         CASE  _response.State 
         OF
           CmdMessageState.BUFFERED : CommandBuffered := TRUE;
           CmdMessageState.DONE     : Done            := TRUE;
           CmdMessageState.ERROR    : Error           := TRUE;
         END_CASE
                
         // Done, Aborted or Error ?
         IF (_response.State >= CmdMessageState.DONE )
         THEN
           // Reset Busy flag
           Busy := FALSE;
           // Update results
           OutCmd.TargetToolNoReturn      := _response.TargetToolNoReturn;
           OutCmd.TargetFrameNoReturn     := _response.TargetFrameNoReturn;
           OutCmd.CartesianPositionReturn := _response.CartesianPositionReturn;

           // set timeout
           SetTimeout(PT := _timeoutCmd, rTimer := _timerCmd);
           // inc step counter
          _stepCmd := _stepCmd + 1; 
         END_IF
       END_IF


  02: IF ( NOT Execute)
      THEN
        Reset();
      END_IF     

ELSE
  // invalid step
  ErrorID := RobotLibraryEvents.ERR_INVALID_STEP;
END_CASE


// Reset FB
IF ( NOT Execute )
THEN
  Reset(); 
END_IF
END_METHOD

METHOD INTERNAL ParseResponsePayload : DINT
VAR_INPUT
  /// Response data
  ResponseData : RobotLibraryRecvDataFB;
  /// Timestamp
  Timestamp    : SystemTime;  
END_VAR
// Table 6-645: Received CMD payload (RC to PLC) of "CalculateCartesianPosition"
// --------------------------
// Header
// --------------------------
// Byte 00 : USINT      - ParSeq | State     
// Byte 01 : SINT       - AlarmMessageSeverity    
// Byte 02 : UINT       - AlarmMessageCode HB
// Byte 03 :            - AlarmMessageCode LB
// --------------------------
// Datablock
// --------------------------
// Byte 04 : USINT      - TargetToolNoReturn
// Byte 05 : USINT      - TargetFrameNoReturn
// Byte 06 : REAL       - Position.X  HW HB
// Byte 07 :            - Position.X  HW LB
// Byte 08 :            - Position.X  LW HB
// Byte 09 :            - Position.X  LW LB
// Byte 10 : REAL       - Position.Y  HW HB
// Byte 11 :            - Position.Y  HW LB
// Byte 12 :            - Position.Y  LW HB
// Byte 13 :            - Position.Y  LW LB
// Byte 14 : REAL       - Position.Z  HW HB
// Byte 15 :            - Position.Z  HW LB
// Byte 16 :            - Position.Z  LW HB
// Byte 17 :            - Position.Z  LW LB
// Byte 18 : REAL       - Position.Rx HW HB
// Byte 19 :            - Position.Rx HW LB
// Byte 20 :            - Position.Rx LW HB
// Byte 21 :            - Position.Rx LW LB
// Byte 22 : REAL       - Position.Ry HW HB
// Byte 23 :            - Position.Ry HW LB
// Byte 24 :            - Position.Ry LW HB
// Byte 25 :            - Position.Ry LW LB
// Byte 26 : REAL       - Position.Rz HW HB
// Byte 27 :            - Position.Rz HW LB
// Byte 28 :            - Position.Rz LW HB
// Byte 29 :            - Position.Rz LW LB
// Byte 30 : Config     - ArmConfig   LW HB
// Byte 31 :            - ArmConfig   LW LB
// Byte 32 : TurnNumber - J1 + J2     LW HB
// Byte 33 :            - J3 + J4     LW LB
// Byte 34 :            - J5 + J6     LW LB
// Byte 35 :            - E1          LW LB
// Byte 36 : REAL       - Position.E1 HW HB
// Byte 37 :            - Position.E1 HW LB
// Byte 38 :            - Position.E1 LW HB
// Byte 39 :            - Position.E1 LW LB
// Byte 40 : REAL       - Position.E2 HW HB
// Byte 41 :            - Position.E2 HW LB
// Byte 42 :            - Position.E2 LW HB
// Byte 43 :            - Position.E2 LW LB
// Byte 44 : REAL       - Position.E3 HW HB
// Byte 45 :            - Position.E3 HW LB
// Byte 46 :            - Position.E3 LW HB
// Byte 47 :            - Position.E3 LW LB
// Byte 48 : REAL       - Position.E4 HW HB
// Byte 49 :            - Position.E4 HW LB
// Byte 50 :            - Position.E4 LW HB
// Byte 51 :            - Position.E4 LW LB
// Byte 52 : REAL       - Position.E5 HW HB
// Byte 53 :            - Position.E5 HW LB
// Byte 54 :            - Position.E5 LW HB
// Byte 55 :            - Position.E5 LW LB
// Byte 56 : REAL       - Position.E6 HW HB
// Byte 57 :            - Position.E6 HW LB
// Byte 58 :            - Position.E6 LW HB
// Byte 59 :            - Position.E6 LW LB
// --------------------------
// call base implementation to parse the header from payload buffer
ResponseData.PayloadPtr := SUPER^.ParseResponsePayload(ResponseData := ResponseData, Timestamp := Timestamp);

// copy parsed header to response
_response.ParSeq               := _rspHeader.ParSeq;
_response.State                := _rspHeader.State;
_response.AlarmMessageSeverity := _rspHeader.AlarmMessageSeverity;
_response.AlarmMessageCode     := _rspHeader.AlarmMessageCode;

// Get TargetToolNoReturn
_response.TargetToolNoReturn   := ResponseData.GetUsint();
// Get TargetFrameNoReturn
_response.TargetFrameNoReturn  := ResponseData.GetUsint();
// Get CartesianPositionReturn.X
_response.CartesianPositionReturn.X := ResponseData.GetReal();
// Get CartesianPositionReturn.Y
_response.CartesianPositionReturn.Y := ResponseData.GetReal();
// Get CartesianPositionReturn.Z
_response.CartesianPositionReturn.Z := ResponseData.GetReal();
// Get CartesianPositionReturn.Rx
_response.CartesianPositionReturn.Rx := ResponseData.GetReal();
// Get CartesianPositionReturn.Ry
_response.CartesianPositionReturn.Ry := ResponseData.GetReal();
// Get CartesianPositionReturn.Rz
_response.CartesianPositionReturn.Rz := ResponseData.GetReal();
// Get CartesianPositionReturn.Config
_response.CartesianPositionReturn.Config := ResponseData.GetArmConfig();
// Get CartesianPositionReturn.TurnNumber
_response.CartesianPositionReturn.TurnNumber := ResponseData.GetTurnNumbers();
// Get CartesianPositionReturn.E1
_response.CartesianPositionReturn.E1 := ResponseData.GetReal();
// Get CartesianPositionReturn.E2
_response.CartesianPositionReturn.E2 := ResponseData.GetReal();
// Get CartesianPositionReturn.E3
_response.CartesianPositionReturn.E3 := ResponseData.GetReal();
// Get CartesianPositionReturn.E4
_response.CartesianPositionReturn.E4 := ResponseData.GetReal();
// Get CartesianPositionReturn.E5
_response.CartesianPositionReturn.E5 := ResponseData.GetReal();
// Get CartesianPositionReturn.E6
_response.CartesianPositionReturn.E6 := ResponseData.GetReal();

// Create logging
ParseResponsePayloadLog(ResponseData := ResponseData, Timestamp := Timestamp);
END_METHOD

METHOD INTERNAL ParseResponsePayloadLog
VAR_INPUT
  /// Response data
  ResponseData : RobotLibraryRecvDataFB;
  /// Timestamp
  Timestamp    : SystemTime;  
END_VAR
// Create log entry for Parameter start
CreateLogMessage      ( Timestamp   := Timestamp,
                        MessageType := MessageType.CMD,
                        Severity    := Severity.DEBUG,
                        MessageCode := 0,
                        MessageText := 'Parsed the following parameter(s) from response data:');
                        
// Create log entry for TargetToolNoReturn
CreateLogMessagePara1 ( Timestamp   := Timestamp,
                        MessageType := MessageType.CMD,
                        Severity    := Severity.DEBUG,
                        MessageCode := 0,
                        MessageText := 'Response.TargetToolNoReturn = {1}',
                        Para1       :=  USINT_TO_STRING(_response.TargetToolNoReturn));

// Create log entry for TargetFrameNoReturn
CreateLogMessagePara1 ( Timestamp   := Timestamp,
                        MessageType := MessageType.CMD,
                        Severity    := Severity.DEBUG,
                        MessageCode := 0,
                        MessageText := 'Response.TargetFrameNoReturn = {1}',
                        Para1       :=  USINT_TO_STRING(_response.TargetFrameNoReturn));

// Create log entry for CartesianPositionReturn.X
CreateLogMessagePara1 ( Timestamp   := Timestamp,
                        MessageType := MessageType.CMD,
                        Severity    := Severity.DEBUG,
                        MessageCode := 0,
                        MessageText := 'Response.CartesianPositionReturn.X = {1}',
                        Para1       :=  REAL_TO_STRING(_response.CartesianPositionReturn.X));

// Create log entry for CartesianPositionReturn.Y
CreateLogMessagePara1 ( Timestamp   := Timestamp,
                        MessageType := MessageType.CMD,
                        Severity    := Severity.DEBUG,
                        MessageCode := 0,
                        MessageText := 'Response.CartesianPositionReturn.Y = {1}',
                        Para1       :=  REAL_TO_STRING(_response.CartesianPositionReturn.Y));

// Create log entry for CartesianPositionReturn.Z
CreateLogMessagePara1 ( Timestamp   := Timestamp,
                        MessageType := MessageType.CMD,
                        Severity    := Severity.DEBUG,
                        MessageCode := 0,
                        MessageText := 'Response.CartesianPositionReturn.Z = {1}',
                        Para1       :=  REAL_TO_STRING(_response.CartesianPositionReturn.Z));

// Create log entry for CartesianPositionReturn.Rx
CreateLogMessagePara1 ( Timestamp   := Timestamp,
                        MessageType := MessageType.CMD,
                        Severity    := Severity.DEBUG,
                        MessageCode := 0,
                        MessageText := 'Response.CartesianPositionReturn.Rx = {1}',
                        Para1       :=  REAL_TO_STRING(_response.CartesianPositionReturn.Rx));

// Create log entry for CartesianPositionReturn.Ry
CreateLogMessagePara1 ( Timestamp   := Timestamp,
                        MessageType := MessageType.CMD,
                        Severity    := Severity.DEBUG,
                        MessageCode := 0,
                        MessageText := 'Response.CartesianPositionReturn.Ry = {1}',
                        Para1       :=  REAL_TO_STRING(_response.CartesianPositionReturn.Ry));

// Create log entry for CartesianPositionReturn.Rz
CreateLogMessagePara1 ( Timestamp   := Timestamp,
                        MessageType := MessageType.CMD,
                        Severity    := Severity.DEBUG,
                        MessageCode := 0,
                        MessageText := 'Response.CartesianPositionReturn.Rz = {1}',
                        Para1       :=  REAL_TO_STRING(_response.CartesianPositionReturn.Rz));

// Create log entry for CartesianPositionReturn.Config
CreateLogMessagePara1 ( Timestamp   := Timestamp,
                        MessageType := MessageType.CMD,
                        Severity    := Severity.DEBUG,
                        MessageCode := 0,
                        MessageText := 'Response.CartesianPositionReturn.Config = {1}',
                        Para1       :=  ARM_CONFIG_TO_STRING(_response.CartesianPositionReturn.Config));

// Create log entry for CartesianPositionReturn.TurnNumber.J1Turns
CreateLogMessagePara1 ( Timestamp   := Timestamp,
                        MessageType := MessageType.CMD,
                        Severity    := Severity.DEBUG,
                        MessageCode := 0,
                        MessageText := 'Response.CartesianPositionReturn.TurnNumber.J1Turns = {1}',
                        Para1       :=  SINT_TO_STRING(_response.CartesianPositionReturn.TurnNumber.J1Turns));

// Create log entry for CartesianPositionReturn.TurnNumber.J2Turns
CreateLogMessagePara1 ( Timestamp   := Timestamp,
                        MessageType := MessageType.CMD,
                        Severity    := Severity.DEBUG,
                        MessageCode := 0,
                        MessageText := 'Response.CartesianPositionReturn.TurnNumber.J2Turns = {1}',
                        Para1       :=  SINT_TO_STRING(_response.CartesianPositionReturn.TurnNumber.J2Turns));

// Create log entry for CartesianPositionReturn.TurnNumber.J3Turns
CreateLogMessagePara1 ( Timestamp   := Timestamp,
                        MessageType := MessageType.CMD,
                        Severity    := Severity.DEBUG,
                        MessageCode := 0,
                        MessageText := 'Response.CartesianPositionReturn.TurnNumber.J3Turns = {1}',
                        Para1       :=  SINT_TO_STRING(_response.CartesianPositionReturn.TurnNumber.J3Turns));

// Create log entry for CartesianPositionReturn.TurnNumber.J4Turns
CreateLogMessagePara1 ( Timestamp   := Timestamp,
                        MessageType := MessageType.CMD,
                        Severity    := Severity.DEBUG,
                        MessageCode := 0,
                        MessageText := 'Response.CartesianPositionReturn.TurnNumber.J4Turns = {1}',
                        Para1       :=  SINT_TO_STRING(_response.CartesianPositionReturn.TurnNumber.J4Turns));

// Create log entry for CartesianPositionReturn.TurnNumber.J5Turns
CreateLogMessagePara1 ( Timestamp   := Timestamp,
                        MessageType := MessageType.CMD,
                        Severity    := Severity.DEBUG,
                        MessageCode := 0,
                        MessageText := 'Response.CartesianPositionReturn.TurnNumber.J5Turns = {1}',
                        Para1       :=  SINT_TO_STRING(_response.CartesianPositionReturn.TurnNumber.J5Turns));

// Create log entry for CartesianPositionReturn.TurnNumber.J6Turns
CreateLogMessagePara1 ( Timestamp   := Timestamp,
                        MessageType := MessageType.CMD,
                        Severity    := Severity.DEBUG,
                        MessageCode := 0,
                        MessageText := 'Response.CartesianPositionReturn.TurnNumber.J6Turns = {1}',
                        Para1       :=  SINT_TO_STRING(_response.CartesianPositionReturn.TurnNumber.J6Turns));

// Create log entry for CartesianPositionReturn.TurnNumber.E1Turns
CreateLogMessagePara1 ( Timestamp   := Timestamp,
                        MessageType := MessageType.CMD,
                        Severity    := Severity.DEBUG,
                        MessageCode := 0,
                        MessageText := 'Response.CartesianPositionReturn.TurnNumber.E1Turns = {1}',
                        Para1       :=  SINT_TO_STRING(_response.CartesianPositionReturn.TurnNumber.E1Turns));

// Create log entry for CartesianPositionReturn.E1
CreateLogMessagePara1 ( Timestamp   := Timestamp,
                        MessageType := MessageType.CMD,
                        Severity    := Severity.DEBUG,
                        MessageCode := 0,
                        MessageText := 'Response.CartesianPositionReturn.E1 = {1}',
                        Para1       :=  REAL_TO_STRING(_response.CartesianPositionReturn.E1));

// Create log entry for CartesianPositionReturn.E2
CreateLogMessagePara1 ( Timestamp   := Timestamp,
                        MessageType := MessageType.CMD,
                        Severity    := Severity.DEBUG,
                        MessageCode := 0,
                        MessageText := 'Response.CartesianPositionReturn.E2 = {1}',
                        Para1       :=  REAL_TO_STRING(_response.CartesianPositionReturn.E2));

// Create log entry for CartesianPositionReturn.E3
CreateLogMessagePara1 ( Timestamp   := Timestamp,
                        MessageType := MessageType.CMD,
                        Severity    := Severity.DEBUG,
                        MessageCode := 0,
                        MessageText := 'Response.CartesianPositionReturn.E3 = {1}',
                        Para1       :=  REAL_TO_STRING(_response.CartesianPositionReturn.E3));

// Create log entry for CartesianPositionReturn.E4
CreateLogMessagePara1 ( Timestamp   := Timestamp,
                        MessageType := MessageType.CMD,
                        Severity    := Severity.DEBUG,
                        MessageCode := 0,
                        MessageText := 'Response.CartesianPositionReturn.E4 = {1}',
                        Para1       :=  REAL_TO_STRING(_response.CartesianPositionReturn.E4));

// Create log entry for CartesianPositionReturn.E5
CreateLogMessagePara1 ( Timestamp   := Timestamp,
                        MessageType := MessageType.CMD,
                        Severity    := Severity.DEBUG,
                        MessageCode := 0,
                        MessageText := 'Response.CartesianPositionReturn.E5 = {1}',
                        Para1       :=  REAL_TO_STRING(_response.CartesianPositionReturn.E5));

// Create log entry for CartesianPositionReturn.E6
CreateLogMessagePara1 ( Timestamp   := Timestamp,
                        MessageType := MessageType.CMD,
                        Severity    := Severity.DEBUG,
                        MessageCode := 0,
                        MessageText := 'Response.CartesianPositionReturn.E6 = {1}',
                        Para1       :=  REAL_TO_STRING(_response.CartesianPositionReturn.E6));
END_METHOD

METHOD PROTECTED Reset : DINT
VAR_INPUT
END_VAR
Reset := SUPER^.Reset();

Done               := FALSE;
Busy               := FALSE;
CommandBuffered    := FALSE;
END_METHOD

END_FUNCTION_BLOCK

// Library/POUs/Calculation/MC_CalculateForwardKinematic/MC_CalculateForwardKinematicFB
/// Calculate Forward Kinematic
FUNCTION_BLOCK MC_CalculateForwardKinematicFB EXTENDS RobotLibraryBaseExecuteFB
// ------------------------------------------------------------------------- 
//  SRCI Robot Library                                                
// ------------------------------------------------------------------------- 
//                                                                           
//  Object:      CalculateForwardKinematicFB                                       
//  Author:      Thorsten Brach                                                
//  Date:        2024-06-01
//
//  Description:                                              
//   
//                                                                           
//  Copyright: 
//    (C) 2024 Thorsten Brach. All rights reserved                                                                                                                                            
//             Licensed under the LGPL-3.0 license.
//                                                                           
//  Disclaimer:                                                                           
//    This project is provided without any guarantee and can be used for   
//    private and commercial purposes. Any use is at the user’s 
//    own risk and responsibility.
//
// -------------------------------------------------------------------------
VAR_INPUT
  /// Command parameter 
  ParCmd          : CalculateForwardKinematicParCmd;    
END_VAR
VAR_OUTPUT
  /// Command is transferred and confirmed by the RC
  CommandBuffered : BOOL;
  /// Command output 
  OutCmd          : CalculateForwardKinematicOutCmd;  
END_VAR

VAR
  /// internal copy of command parameter 
 _parCmd          : CalculateForwardKinematicParCmd;
  /// command data to send
 _command         : CalculateForwardKinematicSendData;
  /// response data received
 _response        : CalculateForwardKinematicRecvData;      
END_VAR

SUPER^(AxesGroup := AxesGroup);

METHOD PROTECTED CheckFunctionSupported : BOOL
VAR_IN_OUT
  /// Robot assignment of function
  AxesGroup : AxesGroup; 
END_VAR
CheckFunctionSupported := AxesGroup.InternalData.RCSupportedFunctions.CalculateForwardKinematic;

IF ( NOT CheckFunctionSupported )
THEN
  // call base implementation for set error and create log entry
  SUPER^.CheckFunctionSupported(AxesGroup := AxesGroup);
END_IF
END_METHOD

METHOD PROTECTED CheckParameterChanged : BOOL
VAR_IN_OUT
  /// Robot assignment of function
  AxesGroup    : AxesGroup; 
END_VAR
// Check ParCmd Size is > 0, because MemCmp does not work correctly with size = 0
IF (SIZEOF(ParCmd) = 0) 
THEN 
  RETURN;
END_IF

// compare memory 
_parameterChanged := ( SysDepMemCmp(pData1 := ADR(ParCmd), pData2 := ADR(_parCmd), DataLen := SIZEOF(ParCmd)) <> RobotLibraryConstants.OK );

// check parameter valid ?
_parameterValid   := CheckParameterValid( AxesGroup := AxesGroup );

IF ((  _parameterChanged        )  AND 
    (  _parameterValid          )) OR
    (  _parameterUpdateInternal )  
THEN  
  // reset internal flag for send parameter update
 _parameterUpdateInternal := FALSE;
  // update internal copy of parameters 
 _parCmd := ParCmd;
  // inc parameter sequence
 _command.ParSeq := _command.ParSeq + 1;
  // update command data  
  CommandData := CreateCommandPayload(AxesGroup := AxesGroup); // ( Access via reference to rCommandFB in ACR )
  // notify active command register 
  AxesGroup.Acyclic.ActiveCommandRegister.NotifyParameterChanged := _uniqueID;
END_IF
END_METHOD

METHOD INTERNAL CreateCommandPayload : RobotLibrarySendDataFB
VAR_IN_OUT
  /// Robot assignment of function
  AxesGroup : AxesGroup; 
END_VAR
// Table 6-632: Sent CMD payload (PLC to RC) of "CalculateForwardKinematic"
// --------------------------
// Header
// --------------------------
// Byte 00 : UINT  - Type HB     
// Byte 01 :       - Type LB    
// Byte 02 : USINT - Reserve | ExecutionMode
// Byte 03 : USINT - ParSeq  | Priority
// --------------------------
// Datablock
// --------------------------
// Byte 04 : USINT - ToolNo
// Byte 05 : USINT - FrameNo
// Byte 06 : REAL  - Position.J1  HW HB
// Byte 07 :       - Position.J1  HW LB
// Byte 08 :       - Position.J1  LW HB
// Byte 09 :       - Position.J1  LW LB
// Byte 10 : REAL  - Position.J2  HW HB
// Byte 11 :       - Position.J2  HW LB
// Byte 12 :       - Position.J2  LW HB
// Byte 13 :       - Position.J2  LW LB
// Byte 14 : REAL  - Position.J3  HW HB
// Byte 15 :       - Position.J3  HW LB
// Byte 16 :       - Position.J3  LW HB
// Byte 17 :       - Position.J3  LW LB
// Byte 18 : REAL  - Position.J4  HW HB
// Byte 19 :       - Position.J4  HW LB
// Byte 20 :       - Position.J4  LW HB
// Byte 21 :       - Position.J4  LW LB
// Byte 22 : REAL  - Position.J5  HW HB
// Byte 23 :       - Position.J5  HW LB
// Byte 24 :       - Position.J5  LW HB
// Byte 25 :       - Position.J5  LW LB
// Byte 26 : REAL  - Position.J6  HW HB
// Byte 27 :       - Position.J6  HW LB
// Byte 28 :       - Position.J6  LW HB
// Byte 29 :       - Position.J6  LW LB
// Byte 30 : REAL  - Position.E1  HW HB
// Byte 31 :       - Position.E1  HW LB
// Byte 32 :       - Position.E1  LW HB
// Byte 33 :       - Position.E1  LW LB
// Byte 34 : REAL  - Position.E2  HW HB
// Byte 35 :       - Position.E2  HW LB
// Byte 36 :       - Position.E2  LW HB
// Byte 37 :       - Position.E2  LW LB
// Byte 38 : REAL  - Position.E3  HW HB
// Byte 39 :       - Position.E3  HW LB
// Byte 40 :       - Position.E3  LW HB
// Byte 41 :       - Position.E3  LW LB
// Byte 42 : REAL  - Position.E4  HW HB
// Byte 43 :       - Position.E4  HW LB
// Byte 44 :       - Position.E4  LW HB
// Byte 45 :       - Position.E4  LW LB
// Byte 46 : REAL  - Position.E5  HW HB
// Byte 47 :       - Position.E5  HW LB
// Byte 48 :       - Position.E5  LW HB
// Byte 49 :       - Position.E5  LW LB
// Byte 50 : REAL  - Position.E6  HW HB
// Byte 51 :       - Position.E6  HW LB
// Byte 52 :       - Position.E6  LW HB
// Byte 53 :       - Position.E6  LW LB

// --------------------------
// set command parameter 
_command.CmdTyp                     :=  CmdType.CalculateForwardKinematic;
_command.ExecMode                   :=  ExecMode;
_command.ParSeq                     := _command.ParSeq;
_command.Priority                   :=  Priority;
_command.ToolNo                     := _parCmd.ToolNo;
_command.FrameNo                    := _parCmd.FrameNo;
_command.JointPosition              := _parCmd.JointPosition;

// copy command data to header
_cmdHeader := _command;
// call base implementation to copy header to payload buffer
CreateCommandPayload := SUPER^.CreateCommandPayload(AxesGroup := AxesGroup);

// add command.ToolNo
CreateCommandPayload.AddUsint(_command.ToolNo);
// add command.FrameNo
CreateCommandPayload.AddUsint(_command.FrameNo);
// add command.JointPosition.J1
CreateCommandPayload.AddReal(_command.JointPosition.J1);
// add command.JointPosition.J2
CreateCommandPayload.AddReal(_command.JointPosition.J2);
// add command.JointPosition.J3
CreateCommandPayload.AddReal(_command.JointPosition.J3);
// add command.JointPosition.J4
CreateCommandPayload.AddReal(_command.JointPosition.J4);
// add command.JointPosition.J5
CreateCommandPayload.AddReal(_command.JointPosition.J5);
// add command.JointPosition.J6
CreateCommandPayload.AddReal(_command.JointPosition.J6);
// add command.JointPosition.E1
CreateCommandPayload.AddReal(_command.JointPosition.E1);
// add command.JointPosition.E2
CreateCommandPayload.AddReal(_command.JointPosition.E2);
// add command.JointPosition.E3
CreateCommandPayload.AddReal(_command.JointPosition.E3);
// add command.JointPosition.E4
CreateCommandPayload.AddReal(_command.JointPosition.E4);
// add command.JointPosition.E5
CreateCommandPayload.AddReal(_command.JointPosition.E5);
// add command.JointPosition.E6
CreateCommandPayload.AddReal(_command.JointPosition.E6);

// Create logging
CreateCommandPayloadLog(AxesGroup := AxesGroup);
END_METHOD

METHOD INTERNAL CreateCommandPayloadLog 
VAR_IN_OUT
  /// Robot assignment of function
  AxesGroup : AxesGroup; 
END_VAR
// Create log entry for Parameter start
CreateLogMessage      ( Timestamp   := AxesGroup.InternalData.SystemTime,
                        MessageType := MessageType.CMD,
                        Severity    := Severity.DEBUG,
                        MessageCode := 0,
                        MessageText := 'Create command payload with the following parameter(s) :');

// Create log entry for ToolNo
CreateLogMessagePara1 ( Timestamp   := AxesGroup.InternalData.SystemTime,
                        MessageType := MessageType.CMD,
                        Severity    := Severity.DEBUG,
                        MessageCode := 0,
                        MessageText := 'Command.ToolNo = {1}',
                        Para1       :=  USINT_TO_STRING(_command.ToolNo));

// Create log entry for FrameNo
CreateLogMessagePara1 ( Timestamp   := AxesGroup.InternalData.SystemTime,
                        MessageType := MessageType.CMD,
                        Severity    := Severity.DEBUG,
                        MessageCode := 0,
                        MessageText := 'Command.FrameNo = {1}',
                        Para1       :=  USINT_TO_STRING(_command.FrameNo));

// Create log entry for JointPosition.J1
CreateLogMessagePara1 ( Timestamp   := AxesGroup.InternalData.SystemTime,
                        MessageType := MessageType.CMD,
                        Severity    := Severity.DEBUG,
                        MessageCode := 0,
                        MessageText := 'Command.JointPosition.J1 = {1}',
                        Para1       :=  REAL_TO_STRING(_command.JointPosition.J1));

// Create log entry for JointPosition.J2
CreateLogMessagePara1 ( Timestamp   := AxesGroup.InternalData.SystemTime,
                        MessageType := MessageType.CMD,
                        Severity    := Severity.DEBUG,
                        MessageCode := 0,
                        MessageText := 'Command.JointPosition.J2 = {1}',
                        Para1       :=  REAL_TO_STRING(_command.JointPosition.J2));

// Create log entry for JointPosition.J3
CreateLogMessagePara1 ( Timestamp   := AxesGroup.InternalData.SystemTime,
                        MessageType := MessageType.CMD,
                        Severity    := Severity.DEBUG,
                        MessageCode := 0,
                        MessageText := 'Command.JointPosition.J3 = {1}',
                        Para1       :=  REAL_TO_STRING(_command.JointPosition.J3));

// Create log entry for JointPosition.J4
CreateLogMessagePara1 ( Timestamp   := AxesGroup.InternalData.SystemTime,
                        MessageType := MessageType.CMD,
                        Severity    := Severity.DEBUG,
                        MessageCode := 0,
                        MessageText := 'Command.JointPosition.J4 = {1}',
                        Para1       :=  REAL_TO_STRING(_command.JointPosition.J4));

// Create log entry for JointPosition.J5
CreateLogMessagePara1 ( Timestamp   := AxesGroup.InternalData.SystemTime,
                        MessageType := MessageType.CMD,
                        Severity    := Severity.DEBUG,
                        MessageCode := 0,
                        MessageText := 'Command.JointPosition.J5 = {1}',
                        Para1       :=  REAL_TO_STRING(_command.JointPosition.J5));

// Create log entry for JointPosition.J6
CreateLogMessagePara1 ( Timestamp   := AxesGroup.InternalData.SystemTime,
                        MessageType := MessageType.CMD,
                        Severity    := Severity.DEBUG,
                        MessageCode := 0,
                        MessageText := 'Command.JointPosition.J6 = {1}',
                        Para1       :=  REAL_TO_STRING(_command.JointPosition.J6));

// Create log entry for JointPosition.E1
CreateLogMessagePara1 ( Timestamp   := AxesGroup.InternalData.SystemTime,
                        MessageType := MessageType.CMD,
                        Severity    := Severity.DEBUG,
                        MessageCode := 0,
                        MessageText := 'Command.JointPosition.E1 = {1}',
                        Para1       :=  REAL_TO_STRING(_command.JointPosition.E1));

// Create log entry for JointPosition.E2
CreateLogMessagePara1 ( Timestamp   := AxesGroup.InternalData.SystemTime,
                        MessageType := MessageType.CMD,
                        Severity    := Severity.DEBUG,
                        MessageCode := 0,
                        MessageText := 'Command.JointPosition.E2 = {1}',
                        Para1       :=  REAL_TO_STRING(_command.JointPosition.E2));

// Create log entry for JointPosition.E3
CreateLogMessagePara1 ( Timestamp   := AxesGroup.InternalData.SystemTime,
                        MessageType := MessageType.CMD,
                        Severity    := Severity.DEBUG,
                        MessageCode := 0,
                        MessageText := 'Command.JointPosition.E3 = {1}',
                        Para1       :=  REAL_TO_STRING(_command.JointPosition.E3));

// Create log entry for JointPosition.E4
CreateLogMessagePara1 ( Timestamp   := AxesGroup.InternalData.SystemTime,
                        MessageType := MessageType.CMD,
                        Severity    := Severity.DEBUG,
                        MessageCode := 0,
                        MessageText := 'Command.JointPosition.E4 = {1}',
                        Para1       :=  REAL_TO_STRING(_command.JointPosition.E4));

// Create log entry for JointPosition.E5
CreateLogMessagePara1 ( Timestamp   := AxesGroup.InternalData.SystemTime,
                        MessageType := MessageType.CMD,
                        Severity    := Severity.DEBUG,
                        MessageCode := 0,
                        MessageText := 'Command.JointPosition.E5 = {1}',
                        Para1       :=  REAL_TO_STRING(_command.JointPosition.E5));

// Create log entry for JointPosition.E6
CreateLogMessagePara1 ( Timestamp   := AxesGroup.InternalData.SystemTime,
                        MessageType := MessageType.CMD,
                        Severity    := Severity.DEBUG,
                        MessageCode := 0,
                        MessageText := 'Command.JointPosition.E6 = {1}',
                        Para1       :=  REAL_TO_STRING(_command.JointPosition.E6));
END_METHOD

METHOD FB_init : BOOL
VAR_INPUT
  /// if TRUE, the retain variables are initialized (warm start / cold start)
  bInitRetains : BOOL; 
  /// if TRUE, the instance afterwards gets moved into the copy code (online change)
  bInCopyCode  : BOOL;  
END_VAR
MyType := 'MC_CalculateForwardKinematicFB';

ExecMode := ExecutionMode.PARALLEL;
END_METHOD

METHOD PROTECTED OnCall
VAR_IN_OUT
  /// Robot assignment of function
  AxesGroup : AxesGroup; 
END_VAR
// call base implementation
SUPER^.OnCall(AxesGroup := AxesGroup);

CASE _stepCmd OF
  
  00:  IF ( _execute_R.Q )  
       THEN
         // Check function is supported and parameter are valid ?
         IF (( CheckFunctionSupported( AxesGroup := AxesGroup )) AND
             ( CheckParameterValid   ( AxesGroup := AxesGroup )))      
         THEN
           // set busy flag
           Busy := TRUE;
           // Reset command outputs
           SysDepMemSet(pDest := ADR(OutCmd), Value := 0, DataLen := SIZEOF(OutCmd));         
           // apply command parameter
          _parCmd := ParCmd;
           // init parameter sequence
          _command.ParSeq := 1;
           // create command data
           CommandData := CreateCommandPayload(AxesGroup := AxesGroup);
           // Add command to active command register
          _uniqueID := AxesGroup.Acyclic.ActiveCommandRegister.AddCmd( pCommandFB := ADR(THIS^ ));     
           // set timeout
           SetTimeout(PT := _timeoutCmd, rTimer := _timerCmd);
           // inc step counter
          _stepCmd := _stepCmd + 1;
         END_IF 
       END_IF
     

  01:  // Wait for responce received
       IF ( _responseReceived )
       THEN
         // reset response received flag
        _responseReceived := FALSE;

         CASE  _response.State 
         OF
           CmdMessageState.BUFFERED : CommandBuffered := TRUE;
           CmdMessageState.DONE     : Error           := TRUE;
           CmdMessageState.ERROR    : Done            := TRUE;
         END_CASE
                
         // Done, Aborted or Error ?
         IF (_response.State >= CmdMessageState.DONE )
         THEN
           // Reset Busy flag
           Busy := FALSE;
           // Update results
           OutCmd.TargetToolNoReturn      := _response.TargetToolNoReturn;
           OutCmd.TargetFrameNoReturn     := _response.TargetFrameNoReturn;
           OutCmd.CartesianPosition       := _response.CartesianPosition;

           // set timeout
           SetTimeout(PT := _timeoutCmd, rTimer := _timerCmd);
           // inc step counter
          _stepCmd := _stepCmd + 1; 
         END_IF
       END_IF


  02: IF ( NOT Execute)
      THEN
        Reset();  
      END_IF     

ELSE
  // invalid step
  ErrorID := RobotLibraryEvents.ERR_INVALID_STEP;
END_CASE


// Reset FB
IF ( NOT Execute )
THEN
  Reset();  
END_IF
END_METHOD

METHOD INTERNAL ParseResponsePayload : DINT
VAR_INPUT
  /// Response data
  ResponseData : RobotLibraryRecvDataFB;
  /// Timestamp
  Timestamp    : SystemTime;  
END_VAR
// Table 6-633: Received CMD payload (RC to PLC) of "CalculateForwardKinematic"
// --------------------------
// Header
// --------------------------
// Byte 00 : USINT      - ParSeq | State     
// Byte 01 : SINT       - AlarmMessageSeverity    
// Byte 02 : UINT       - AlarmMessageCode HB
// Byte 03 :            - AlarmMessageCode LB
// --------------------------
// Datablock
// --------------------------
// Byte 04 : USINT      - ToolNoReturn
// Byte 05 : USINT      - FrameNoReturn
// Byte 06 : REAL       - Position.X  HW HB
// Byte 07 :            - Position.X  HW LB
// Byte 08 :            - Position.X  LW HB
// Byte 09 :            - Position.X  LW LB
// Byte 10 : REAL       - Position.Y  HW HB
// Byte 11 :            - Position.Y  HW LB
// Byte 12 :            - Position.Y  LW HB
// Byte 13 :            - Position.Y  LW LB
// Byte 14 : REAL       - Position.Z  HW HB
// Byte 15 :            - Position.Z  HW LB
// Byte 16 :            - Position.Z  LW HB
// Byte 17 :            - Position.Z  LW LB
// Byte 18 : REAL       - Position.Rx HW HB
// Byte 19 :            - Position.Rx HW LB
// Byte 20 :            - Position.Rx LW HB
// Byte 21 :            - Position.Rx LW LB
// Byte 22 : REAL       - Position.Ry HW HB
// Byte 23 :            - Position.Ry HW LB
// Byte 24 :            - Position.Ry LW HB
// Byte 25 :            - Position.Ry LW LB
// Byte 26 : REAL       - Position.Rz HW HB
// Byte 27 :            - Position.Rz HW LB
// Byte 28 :            - Position.Rz LW HB
// Byte 29 :            - Position.Rz LW LB
// Byte 30 : Config     - ArmConfig   LW HB
// Byte 31 :            - ArmConfig   LW LB
// Byte 32 : TurnNumber - J1 + J2     LW HB
// Byte 33 :            - J3 + J4     LW LB
// Byte 34 :            - J5 + J6     LW LB
// Byte 35 :            - E1          LW LB
// Byte 36 : REAL       - Position.E1 HW HB
// Byte 37 :            - Position.E1 HW LB
// Byte 38 :            - Position.E1 LW HB
// Byte 39 :            - Position.E1 LW LB
// Byte 40 : REAL       - Position.E2 HW HB
// Byte 41 :            - Position.E2 HW LB
// Byte 42 :            - Position.E2 LW HB
// Byte 43 :            - Position.E2 LW LB
// Byte 44 : REAL       - Position.E3 HW HB
// Byte 45 :            - Position.E3 HW LB
// Byte 46 :            - Position.E3 LW HB
// Byte 47 :            - Position.E3 LW LB
// Byte 48 : REAL       - Position.E4 HW HB
// Byte 49 :            - Position.E4 HW LB
// Byte 50 :            - Position.E4 LW HB
// Byte 51 :            - Position.E4 LW LB
// Byte 52 : REAL       - Position.E5 HW HB
// Byte 53 :            - Position.E5 HW LB
// Byte 54 :            - Position.E5 LW HB
// Byte 55 :            - Position.E5 LW LB
// Byte 56 : REAL       - Position.E6 HW HB
// Byte 57 :            - Position.E6 HW LB
// Byte 58 :            - Position.E6 LW HB
// Byte 59 :            - Position.E6 LW LB
// --------------------------
// call base implementation to parse the header from payload buffer
ResponseData.PayloadPtr := SUPER^.ParseResponsePayload(ResponseData := ResponseData, Timestamp := Timestamp);

// copy parsed header to response
_response.ParSeq               := _rspHeader.ParSeq;
_response.State                := _rspHeader.State;
_response.AlarmMessageSeverity := _rspHeader.AlarmMessageSeverity;
_response.AlarmMessageCode     := _rspHeader.AlarmMessageCode;

// Get TargetToolNoReturn
_response.TargetToolNoReturn   := ResponseData.GetUsint();
// Get TargetFrameNoReturn
_response.TargetFrameNoReturn  := ResponseData.GetUsint();
// Get CartesianPosition.X
_response.CartesianPosition.X := ResponseData.GetReal();
// Get CartesianPosition.Y
_response.CartesianPosition.Y := ResponseData.GetReal();
// Get CartesianPosition.Z
_response.CartesianPosition.Z := ResponseData.GetReal();
// Get CartesianPosition.Rx
_response.CartesianPosition.Rx := ResponseData.GetReal();
// Get CartesianPosition.Ry
_response.CartesianPosition.Ry := ResponseData.GetReal();
// Get CartesianPosition.Rz
_response.CartesianPosition.Rz := ResponseData.GetReal();
// Get CartesianPosition.Config
_response.CartesianPosition.Config := ResponseData.GetArmConfig();
// Get CartesianPosition.TurnNumber
_response.CartesianPosition.TurnNumber := ResponseData.GetTurnNumbers();
// Get CartesianPosition.E1
_response.CartesianPosition.E1 := ResponseData.GetReal();
// Get CartesianPosition.E2
_response.CartesianPosition.E2 := ResponseData.GetReal();
// Get CartesianPosition.E3
_response.CartesianPosition.E3 := ResponseData.GetReal();
// Get CartesianPosition.E4
_response.CartesianPosition.E4 := ResponseData.GetReal();
// Get CartesianPosition.E5
_response.CartesianPosition.E5 := ResponseData.GetReal();
// Get CartesianPosition.E6
_response.CartesianPosition.E6 := ResponseData.GetReal();

// Create logging
ParseResponsePayloadLog(ResponseData := ResponseData, Timestamp := Timestamp);
END_METHOD

METHOD INTERNAL ParseResponsePayloadLog
VAR_INPUT
  /// Response data
  ResponseData : RobotLibraryRecvDataFB;
  /// Timestamp
  Timestamp    : SystemTime;  
END_VAR
// Create log entry for Parameter start
CreateLogMessage      ( Timestamp   := Timestamp,
                        MessageType := MessageType.CMD,
                        Severity    := Severity.DEBUG,
                        MessageCode := 0,
                        MessageText := 'Parsed the following parameter(s) from response data:');
                        
// Create log entry for TargetToolNoReturn
CreateLogMessagePara1 ( Timestamp   := Timestamp,
                        MessageType := MessageType.CMD,
                        Severity    := Severity.DEBUG,
                        MessageCode := 0,
                        MessageText := 'Response.TargetToolNoReturn = {1}',
                        Para1       :=  USINT_TO_STRING(_response.TargetToolNoReturn));

// Create log entry for TargetFrameNoReturn
CreateLogMessagePara1 ( Timestamp   := Timestamp,
                        MessageType := MessageType.CMD,
                        Severity    := Severity.DEBUG,
                        MessageCode := 0,
                        MessageText := 'Response.TargetFrameNoReturn = {1}',
                        Para1       :=  USINT_TO_STRING(_response.TargetFrameNoReturn));

// Create log entry for CartesianPosition.X
CreateLogMessagePara1 ( Timestamp   := Timestamp,
                        MessageType := MessageType.CMD,
                        Severity    := Severity.DEBUG,
                        MessageCode := 0,
                        MessageText := 'Response.CartesianPosition.X = {1}',
                        Para1       :=  REAL_TO_STRING(_response.CartesianPosition.X));

// Create log entry for CartesianPosition.Y
CreateLogMessagePara1 ( Timestamp   := Timestamp,
                        MessageType := MessageType.CMD,
                        Severity    := Severity.DEBUG,
                        MessageCode := 0,
                        MessageText := 'Response.CartesianPosition.Y = {1}',
                        Para1       :=  REAL_TO_STRING(_response.CartesianPosition.Y));

// Create log entry for CartesianPosition.Z
CreateLogMessagePara1 ( Timestamp   := Timestamp,
                        MessageType := MessageType.CMD,
                        Severity    := Severity.DEBUG,
                        MessageCode := 0,
                        MessageText := 'Response.CartesianPosition.Z = {1}',
                        Para1       :=  REAL_TO_STRING(_response.CartesianPosition.Z));

// Create log entry for CartesianPosition.Rx
CreateLogMessagePara1 ( Timestamp   := Timestamp,
                        MessageType := MessageType.CMD,
                        Severity    := Severity.DEBUG,
                        MessageCode := 0,
                        MessageText := 'Response.CartesianPosition.Rx = {1}',
                        Para1       :=  REAL_TO_STRING(_response.CartesianPosition.Rx));

// Create log entry for CartesianPosition.Ry
CreateLogMessagePara1 ( Timestamp   := Timestamp,
                        MessageType := MessageType.CMD,
                        Severity    := Severity.DEBUG,
                        MessageCode := 0,
                        MessageText := 'Response.CartesianPosition.Ry = {1}',
                        Para1       :=  REAL_TO_STRING(_response.CartesianPosition.Ry));

// Create log entry for CartesianPosition.Rz
CreateLogMessagePara1 ( Timestamp   := Timestamp,
                        MessageType := MessageType.CMD,
                        Severity    := Severity.DEBUG,
                        MessageCode := 0,
                        MessageText := 'Response.CartesianPosition.Rz = {1}',
                        Para1       :=  REAL_TO_STRING(_response.CartesianPosition.Rz));

// Create log entry for CartesianPosition.Config
CreateLogMessagePara1 ( Timestamp   := Timestamp,
                        MessageType := MessageType.CMD,
                        Severity    := Severity.DEBUG,
                        MessageCode := 0,
                        MessageText := 'Response.CartesianPosition.Config = {1}',
                        Para1       :=  ARM_CONFIG_TO_STRING(_response.CartesianPosition.Config));

// Create log entry for CartesianPosition.TurnNumber.J1Turns
CreateLogMessagePara1 ( Timestamp   := Timestamp,
                        MessageType := MessageType.CMD,
                        Severity    := Severity.DEBUG,
                        MessageCode := 0,
                        MessageText := 'Response.CartesianPosition.TurnNumber.J1Turns = {1}',
                        Para1       :=  SINT_TO_STRING(_response.CartesianPosition.TurnNumber.J1Turns));

// Create log entry for CartesianPosition.TurnNumber.J2Turns
CreateLogMessagePara1 ( Timestamp   := Timestamp,
                        MessageType := MessageType.CMD,
                        Severity    := Severity.DEBUG,
                        MessageCode := 0,
                        MessageText := 'Response.CartesianPosition.TurnNumber.J2Turns = {1}',
                        Para1       :=  SINT_TO_STRING(_response.CartesianPosition.TurnNumber.J2Turns));

// Create log entry for CartesianPosition.TurnNumber.J3Turns
CreateLogMessagePara1 ( Timestamp   := Timestamp,
                        MessageType := MessageType.CMD,
                        Severity    := Severity.DEBUG,
                        MessageCode := 0,
                        MessageText := 'Response.CartesianPosition.TurnNumber.J3Turns = {1}',
                        Para1       :=  SINT_TO_STRING(_response.CartesianPosition.TurnNumber.J3Turns));

// Create log entry for CartesianPosition.TurnNumber.J4Turns
CreateLogMessagePara1 ( Timestamp   := Timestamp,
                        MessageType := MessageType.CMD,
                        Severity    := Severity.DEBUG,
                        MessageCode := 0,
                        MessageText := 'Response.CartesianPosition.TurnNumber.J4Turns = {1}',
                        Para1       :=  SINT_TO_STRING(_response.CartesianPosition.TurnNumber.J4Turns));

// Create log entry for CartesianPosition.TurnNumber.J5Turns
CreateLogMessagePara1 ( Timestamp   := Timestamp,
                        MessageType := MessageType.CMD,
                        Severity    := Severity.DEBUG,
                        MessageCode := 0,
                        MessageText := 'Response.CartesianPosition.TurnNumber.J5Turns = {1}',
                        Para1       :=  SINT_TO_STRING(_response.CartesianPosition.TurnNumber.J5Turns));

// Create log entry for CartesianPosition.TurnNumber.J6Turns
CreateLogMessagePara1 ( Timestamp   := Timestamp,
                        MessageType := MessageType.CMD,
                        Severity    := Severity.DEBUG,
                        MessageCode := 0,
                        MessageText := 'Response.CartesianPosition.TurnNumber.J6Turns = {1}',
                        Para1       :=  SINT_TO_STRING(_response.CartesianPosition.TurnNumber.J6Turns));

// Create log entry for CartesianPosition.TurnNumber.E1Turns
CreateLogMessagePara1 ( Timestamp   := Timestamp,
                        MessageType := MessageType.CMD,
                        Severity    := Severity.DEBUG,
                        MessageCode := 0,
                        MessageText := 'Response.CartesianPosition.TurnNumber.E1Turns = {1}',
                        Para1       :=  SINT_TO_STRING(_response.CartesianPosition.TurnNumber.E1Turns));

// Create log entry for CartesianPosition.E1
CreateLogMessagePara1 ( Timestamp   := Timestamp,
                        MessageType := MessageType.CMD,
                        Severity    := Severity.DEBUG,
                        MessageCode := 0,
                        MessageText := 'Response.CartesianPosition.E1 = {1}',
                        Para1       :=  REAL_TO_STRING(_response.CartesianPosition.E1));

// Create log entry for CartesianPosition.E2
CreateLogMessagePara1 ( Timestamp   := Timestamp,
                        MessageType := MessageType.CMD,
                        Severity    := Severity.DEBUG,
                        MessageCode := 0,
                        MessageText := 'Response.CartesianPosition.E2 = {1}',
                        Para1       :=  REAL_TO_STRING(_response.CartesianPosition.E2));

// Create log entry for CartesianPosition.E3
CreateLogMessagePara1 ( Timestamp   := Timestamp,
                        MessageType := MessageType.CMD,
                        Severity    := Severity.DEBUG,
                        MessageCode := 0,
                        MessageText := 'Response.CartesianPosition.E3 = {1}',
                        Para1       :=  REAL_TO_STRING(_response.CartesianPosition.E3));

// Create log entry for CartesianPosition.E4
CreateLogMessagePara1 ( Timestamp   := Timestamp,
                        MessageType := MessageType.CMD,
                        Severity    := Severity.DEBUG,
                        MessageCode := 0,
                        MessageText := 'Response.CartesianPosition.E4 = {1}',
                        Para1       :=  REAL_TO_STRING(_response.CartesianPosition.E4));

// Create log entry for CartesianPosition.E5
CreateLogMessagePara1 ( Timestamp   := Timestamp,
                        MessageType := MessageType.CMD,
                        Severity    := Severity.DEBUG,
                        MessageCode := 0,
                        MessageText := 'Response.CartesianPosition.E5 = {1}',
                        Para1       :=  REAL_TO_STRING(_response.CartesianPosition.E5));

// Create log entry for CartesianPosition.E6
CreateLogMessagePara1 ( Timestamp   := Timestamp,
                        MessageType := MessageType.CMD,
                        Severity    := Severity.DEBUG,
                        MessageCode := 0,
                        MessageText := 'Response.CartesianPosition.E6 = {1}',
                        Para1       :=  REAL_TO_STRING(_response.CartesianPosition.E6));
END_METHOD

METHOD PROTECTED Reset : DINT
VAR_INPUT
END_VAR
Reset := SUPER^.Reset();

Done               := FALSE;
Busy               := FALSE;
CommandBuffered    := FALSE;
END_METHOD

END_FUNCTION_BLOCK

// Library/POUs/Calculation/MC_CalculateFrame/MC_CalculateFrameFB
/// Calculate frame with three-point method
FUNCTION_BLOCK MC_CalculateFrameFB EXTENDS RobotLibraryBaseExecuteFB
// ------------------------------------------------------------------------- 
//  SRCI Robot Library                                                
// ------------------------------------------------------------------------- 
//                                                                           
//  Object:      CalculateFrameFB                                       
//  Author:      Thorsten Brach                                                
//  Date:        2024-06-09
//
//  Description:                                              
//   
//                                                                           
//  Copyright: 
//    (C) 2024 Thorsten Brach. All rights reserved                                                                                                                                            
//             Licensed under the LGPL-3.0 license.
//                                                                           
//  Disclaimer:                                                                           
//    This project is provided without any guarantee and can be used for   
//    private and commercial purposes. Any use is at the user’s 
//    own risk and responsibility.
//
// -------------------------------------------------------------------------
VAR_INPUT
  /// command parameter 
  ParCmd          : CalculateFrameParCmd;
END_VAR
VAR_OUTPUT
  /// Command is transferred and confirmed by the RC
  CommandBuffered : BOOL;
  /// Command output 
  OutCmd          : CalculateFrameOutCmd;    
END_VAR

VAR
  /// internal copy of command parameter 
 _parCmd          : CalculateFrameParCmd;
  /// command data to send
 _command         : CalculateFrameSendData;
  /// response data received
 _response        : CalculateFrameRecvData;      
  /// Incremented with each position of the input parameter "PositionsArray" sent from the PLC to the RC.
  /// Default: 0
 _dataIndex       : USINT;
  /// Set TRUE by the client, when according to the user selected "Mode" the final position of the input parameter "PositionsArray" is sent to the RC.
  /// Default: FALSE
 _dataComplete    : BOOL;
END_VAR

SUPER^(AxesGroup := AxesGroup);

METHOD PROTECTED CheckFunctionSupported : BOOL
VAR_IN_OUT
  /// Robot assignment of function
  AxesGroup : AxesGroup; 
END_VAR
CheckFunctionSupported := AxesGroup.InternalData.RCSupportedFunctions.CalculateFrame;

IF ( NOT CheckFunctionSupported )
THEN
  // call base implementation for set error and create log entry
  SUPER^.CheckFunctionSupported(AxesGroup := AxesGroup);
END_IF
END_METHOD

METHOD PROTECTED CheckParameterChanged : BOOL
VAR_IN_OUT
  /// Robot assignment of function
  AxesGroup    : AxesGroup; 
END_VAR
// Check ParCmd Size is > 0, because MemCmp does not work correctly with size = 0
IF (SIZEOF(ParCmd) = 0) 
THEN 
  RETURN;
END_IF

// compare memory 
_parameterChanged := ( SysDepMemCmp(pData1 := ADR(ParCmd), pData2 := ADR(_parCmd), DataLen := SIZEOF(ParCmd)) <> RobotLibraryConstants.OK );

// check parameter valid ?
_parameterValid   := CheckParameterValid( AxesGroup := AxesGroup );

IF ((  _parameterChanged        )  AND 
    (  _parameterValid          )) OR
    (  _parameterUpdateInternal )  
THEN  
  // reset internal flag for send parameter update
 _parameterUpdateInternal := FALSE;
  // update internal copy of parameters 
 _parCmd := ParCmd;
  // inc parameter sequence
 _command.ParSeq := _command.ParSeq + 1;
  // update command data  
  CommandData := CreateCommandPayload(AxesGroup := AxesGroup); // ( Access via reference to rCommandFB in ACR )
  // notify active command register 
  AxesGroup.Acyclic.ActiveCommandRegister.NotifyParameterChanged := _uniqueID;
END_IF
END_METHOD

METHOD INTERNAL CreateCommandPayload : RobotLibrarySendDataFB
VAR_IN_OUT
  /// Robot assignment of function
  AxesGroup : AxesGroup; 
END_VAR
// Table 6-656: Sent CMD payload (PLC to RC) of "CalculateFrame"
// --------------------------
// Header
// --------------------------
// Byte 00 : UINT       - Type HB     
// Byte 01 :            - Type LB    
// Byte 02 : USINT      - Reserve | ExecutionMode
// Byte 03 : USINT      - ParSeq  | Priority
// --------------------------
// Datablock
// --------------------------
// Byte 04 : USIN       - DataIndex
// Byte 05 : BOOL       - DataComplete
// Byte 06 : BYTE       - Reserve
// Byte 07 : USINT      - FrameNo
// Byte 08 : USINT      - ReferenceFrame
// Byte 09 : SINT       - Mode
// Byte 10 : REAL       - Position X  HW HB
// Byte 11 :            - Position X  HW LB
// Byte 12 :            - Position X  LW HB
// Byte 13 :            - Position X  LW LB
// Byte 14 : REAL       - Position Y  HW HB
// Byte 15 :            - Position Y  HW LB
// Byte 16 :            - Position Y  LW HB
// Byte 17 :            - Position Y  LW LB
// Byte 18 : REAL       - Position Z  HW HB
// Byte 19 :            - Position Z  HW LB
// Byte 20 :            - Position Z  LW HB
// Byte 21 :            - Position Z  LW LB
// Byte 22 : REAL       - Position Rx HW HB
// Byte 23 :            - Position Rx HW LB
// Byte 24 :            - Position Rx LW HB
// Byte 25 :            - Position Rx LW LB
// Byte 26 : REAL       - Position Ry HW HB
// Byte 27 :            - Position Ry HW LB
// Byte 28 :            - Position Ry LW HB
// Byte 29 :            - Position Ry LW LB
// Byte 30 : REAL       - Position Rz HW HB
// Byte 31 :            - Position Rz HW LB
// Byte 32 :            - Position Rz LW HB
// Byte 33 :            - Position Rz LW LB
// Byte 34 : Config     - ArmConfig   LW HB
// Byte 35 :            - ArmConfig   LW LB
// Byte 36 : TurnNumber - J1 + J2     LW HB
// Byte 37 :            - J3 + J4     LW LB
// Byte 38 :            - J5 + J6     LW LB
// Byte 39 :            - E1          LW LB
// Byte 40 : REAL       - Position E1 HW HB
// Byte 41 :            - Position E1 HW LB
// Byte 42 :            - Position E1 LW HB
// Byte 43 :            - Position E1 LW LB
// Byte 44 : REAL       - Position E2 HW HB
// Byte 45 :            - Position E2 HW LB
// Byte 46 :            - Position E2 LW HB
// Byte 47 :            - Position E2 LW LB
// Byte 48 : REAL       - Position E3 HW HB
// Byte 49 :            - Position E3 HW LB
// Byte 50 :            - Position E3 LW HB
// Byte 51 :            - Position E3 LW LB
// Byte 52 : REAL       - Position E4 HW HB
// Byte 53 :            - Position E4 HW LB
// Byte 54 :            - Position E4 LW HB
// Byte 55 :            - Position E4 LW LB
// Byte 56 : REAL       - Position E5 HW HB
// Byte 57 :            - Position E5 HW LB
// Byte 58 :            - Position E5 LW HB
// Byte 59 :            - Position E5 LW LB
// Byte 60 : REAL       - Position E6 HW HB
// Byte 61 :            - Position E6 HW LB
// Byte 62 :            - Position E6 LW HB
// Byte 63 :            - Position E6 LW LB
// --------------------------
// set command parameter 
_command.CmdTyp         :=  CmdType.CalculateFrame;
_command.ExecMode       :=  ExecMode;
_command.ParSeq         := _command.ParSeq;
_command.Priority       :=  Priority;
_command.FrameNo        := _parCmd.FrameNo;
_command.DataIndex      := _dataIndex;
_command.DataComplete.0 := _dataComplete;
_command.Reserve        := 0;
_command.FrameNo        := _parCmd.FrameNo;                 
_command.ReferenceFrame := _parCmd.ReferenceFrame;
_command.Mode           := _parCmd.Mode;

CASE _parCmd.Mode OF
  
  FrameCalculationMode.THREE_POINT_METHOD :

    CASE _dataIndex OF
      
      1: _command.Position := _parCmd.Origin;
      2: _command.Position := _parCmd.Position_X;
      3: _command.Position := _parCmd.Position_XY;
      
    END_CASE
  
  FrameCalculationMode.FOUR_POINT_METHOD  :

    CASE _dataIndex OF
      
      1: _command.Position := _parCmd.Origin;
      2: _command.Position := _parCmd.Position_X;
      3: _command.Position := _parCmd.Position_XY;
      4: _command.Position := _parCmd.OriginShift;      

    END_CASE
  
  FrameCalculationMode.ONE_POINT_METHOD   :
  
   _command.Position := _parCmd.Origin;

END_CASE

// copy command data to header
_cmdHeader := _command;
// call base implementation to copy header to payload buffer
CreateCommandPayload := SUPER^.CreateCommandPayload(AxesGroup := AxesGroup);

// add command.DataIndex
CreateCommandPayload.AddUsint(_command.DataIndex);
// add command.DataComplete
CreateCommandPayload.AddByte(_command.DataComplete);
// add command.Reserve
CreateCommandPayload.AddByte(_command.Reserve);
// add command.FrameNo
CreateCommandPayload.AddUsint(_command.FrameNo);
// add command.ReferenceFrame
CreateCommandPayload.AddUsint(_command.ReferenceFrame);
// add command.Mode
CreateCommandPayload.AddSint(_command.Mode);
// add command.Position.X
CreateCommandPayload.AddReal(_command.Position.X);
// add command.Position.Y
CreateCommandPayload.AddReal(_command.Position.Y);
// add command.Position.Z
CreateCommandPayload.AddReal(_command.Position.Z);
// add command.Position.Rx
CreateCommandPayload.AddReal(_command.Position.Rx);
// add command.Position.Ry
CreateCommandPayload.AddReal(_command.Position.Ry);
// add command.Position.Rz
CreateCommandPayload.AddReal(_command.Position.Rz);
// add command.Position.Config
CreateCommandPayload.AddArmConfig(_command.Position.Config);
// add command.Position.TurnNumber
CreateCommandPayload.AddTurnNumber(_command.Position.TurnNumber);
// add command.Position.E1
CreateCommandPayload.AddReal(_command.Position.E1);
// add command.Position.E2
CreateCommandPayload.AddReal(_command.Position.E2);
// add command.Position.E3
CreateCommandPayload.AddReal(_command.Position.E3);
// add command.Position.E4
CreateCommandPayload.AddReal(_command.Position.E4);
// add command.Position.E5
CreateCommandPayload.AddReal(_command.Position.E5);
// add command.Position.E6
CreateCommandPayload.AddReal(_command.Position.E6);

// Create logging
CreateCommandPayloadLog(AxesGroup := AxesGroup);
END_METHOD

METHOD INTERNAL CreateCommandPayloadLog 
VAR_IN_OUT
  /// Robot assignment of function
  AxesGroup : AxesGroup; 
END_VAR
// Create log entry for Parameter start
CreateLogMessage      ( Timestamp   := AxesGroup.InternalData.SystemTime,
                        MessageType := MessageType.CMD,
                        Severity    := Severity.DEBUG,
                        MessageCode := 0,
                        MessageText := 'Create command payload with the following parameter(s) :');

// Create log entry for DataIndex
CreateLogMessagePara1 ( Timestamp   := AxesGroup.InternalData.SystemTime,
                        MessageType := MessageType.CMD,
                        Severity    := Severity.DEBUG,
                        MessageCode := 0,
                        MessageText := 'Command.DataIndex = {1}',
                        Para1       :=  USINT_TO_STRING(_command.DataIndex));

// Create log entry for DataComplete
CreateLogMessagePara1 ( Timestamp   := AxesGroup.InternalData.SystemTime,
                        MessageType := MessageType.CMD,
                        Severity    := Severity.DEBUG,
                        MessageCode := 0,
                        MessageText := 'Command.DataComplete = {1}',
                        Para1       :=  BYTE_TO_STRING(_command.DataComplete));

// Create log entry for Reserve
CreateLogMessagePara1 ( Timestamp   := AxesGroup.InternalData.SystemTime,
                        MessageType := MessageType.CMD,
                        Severity    := Severity.DEBUG,
                        MessageCode := 0,
                        MessageText := 'Command.Reserve = {1}',
                        Para1       :=  BYTE_TO_STRING(_command.Reserve));

// Create log entry for FrameNo
CreateLogMessagePara1 ( Timestamp   := AxesGroup.InternalData.SystemTime,
                        MessageType := MessageType.CMD,
                        Severity    := Severity.DEBUG,
                        MessageCode := 0,
                        MessageText := 'Command.FrameNo = {1}',
                        Para1       :=  USINT_TO_STRING(_command.FrameNo));

// Create log entry for ReferenceFrame
CreateLogMessagePara1 ( Timestamp   := AxesGroup.InternalData.SystemTime,
                        MessageType := MessageType.CMD,
                        Severity    := Severity.DEBUG,
                        MessageCode := 0,
                        MessageText := 'Command.ReferenceFrame = {1}',
                        Para1       :=  USINT_TO_STRING(_command.ReferenceFrame));

// Create log entry for Mode
CreateLogMessagePara1 ( Timestamp   := AxesGroup.InternalData.SystemTime,
                        MessageType := MessageType.CMD,
                        Severity    := Severity.DEBUG,
                        MessageCode := 0,
                        MessageText := 'Command.Mode = {1}',
                        Para1       :=  FRAME_CALCULATION_MODE_TO_STRING(_command.Mode));


// Create log entry for Position.X
CreateLogMessagePara1 ( Timestamp   := AxesGroup.InternalData.SystemTime,
                        MessageType := MessageType.CMD,
                        Severity    := Severity.DEBUG,
                        MessageCode := 0,
                        MessageText := 'Command.Position.X = {1}',
                        Para1       :=  REAL_TO_STRING(_command.Position.X));

// Create log entry for Position.Y
CreateLogMessagePara1 ( Timestamp   := AxesGroup.InternalData.SystemTime,
                        MessageType := MessageType.CMD,
                        Severity    := Severity.DEBUG,
                        MessageCode := 0,
                        MessageText := 'Command.Position.Y = {1}',
                        Para1       :=  REAL_TO_STRING(_command.Position.Y));

// Create log entry for Position.Z
CreateLogMessagePara1 ( Timestamp   := AxesGroup.InternalData.SystemTime,
                        MessageType := MessageType.CMD,
                        Severity    := Severity.DEBUG,
                        MessageCode := 0,
                        MessageText := 'Command.Position.Z = {1}',
                        Para1       :=  REAL_TO_STRING(_command.Position.Z));

// Create log entry for Position.Rx
CreateLogMessagePara1 ( Timestamp   := AxesGroup.InternalData.SystemTime,
                        MessageType := MessageType.CMD,
                        Severity    := Severity.DEBUG,
                        MessageCode := 0,
                        MessageText := 'Command.Position.Rx = {1}',
                        Para1       :=  REAL_TO_STRING(_command.Position.Rx));

// Create log entry for Position.Ry
CreateLogMessagePara1 ( Timestamp   := AxesGroup.InternalData.SystemTime,
                        MessageType := MessageType.CMD,
                        Severity    := Severity.DEBUG,
                        MessageCode := 0,
                        MessageText := 'Command.Position.Ry = {1}',
                        Para1       :=  REAL_TO_STRING(_command.Position.Ry));

// Create log entry for Position.Rz
CreateLogMessagePara1 ( Timestamp   := AxesGroup.InternalData.SystemTime,
                        MessageType := MessageType.CMD,
                        Severity    := Severity.DEBUG,
                        MessageCode := 0,
                        MessageText := 'Command.Position.Rz = {1}',
                        Para1       :=  REAL_TO_STRING(_command.Position.Rz));

// Create log entry for Position.Config
CreateLogMessagePara1 ( Timestamp   := AxesGroup.InternalData.SystemTime,
                        MessageType := MessageType.CMD,
                        Severity    := Severity.DEBUG,
                        MessageCode := 0,
                        MessageText := 'Command.Position.Config = {1}',
                        Para1       :=  ARM_CONFIG_TO_STRING(_command.Position.Config));

// Create log entry for Position.TurnNumber[0]
CreateLogMessagePara1 ( Timestamp   := AxesGroup.InternalData.SystemTime,
                        MessageType := MessageType.CMD,
                        Severity    := Severity.DEBUG,
                        MessageCode := 0,
                        MessageText := 'Command.Position.TurnNumber[0] = {1}',
                        Para1       :=  BYTE_TO_STRING(CombineHalfSints(HalfSintHi := _command.Position.TurnNumber.J2Turns, 
                                                                        HalfSintLo := _command.Position.TurnNumber.J1Turns)));

// Create log entry for Position.TurnNumber[1]
CreateLogMessagePara1 ( Timestamp   := AxesGroup.InternalData.SystemTime,
                        MessageType := MessageType.CMD,
                        Severity    := Severity.DEBUG,
                        MessageCode := 0,
                        MessageText := 'Command.Position.TurnNumber[1] = {1}',
                        Para1       :=  BYTE_TO_STRING(CombineHalfSints(HalfSintHi := _command.Position.TurnNumber.J4Turns, 
                                                                        HalfSintLo := _command.Position.TurnNumber.J3Turns)));

// Create log entry for Position.TurnNumber[2]
CreateLogMessagePara1 ( Timestamp   := AxesGroup.InternalData.SystemTime,
                        MessageType := MessageType.CMD,
                        Severity    := Severity.DEBUG,
                        MessageCode := 0,
                        MessageText := 'Command.Position.TurnNumber[2] = {1}',
                        Para1       :=  BYTE_TO_STRING(CombineHalfSints(HalfSintHi := _command.Position.TurnNumber.J6Turns, 
                                                                        HalfSintLo := _command.Position.TurnNumber.J5Turns)));

// Create log entry for Position.TurnNumber[3]
CreateLogMessagePara1 ( Timestamp   := AxesGroup.InternalData.SystemTime,
                        MessageType := MessageType.CMD,
                        Severity    := Severity.DEBUG,
                        MessageCode := 0,
                        MessageText := 'Command.Position.TurnNumber[3] = {1}',
                        Para1       :=  SINT_TO_STRING(_command.Position.TurnNumber.E1Turns));

// Create log entry for Position.E1
CreateLogMessagePara1 ( Timestamp   := AxesGroup.InternalData.SystemTime,
                        MessageType := MessageType.CMD,
                        Severity    := Severity.DEBUG,
                        MessageCode := 0,
                        MessageText := 'Command.Position.E1 = {1}',
                        Para1       :=  REAL_TO_STRING(_command.Position.E1));

// Create log entry for Position.E2
CreateLogMessagePara1 ( Timestamp   := AxesGroup.InternalData.SystemTime,
                        MessageType := MessageType.CMD,
                        Severity    := Severity.DEBUG,
                        MessageCode := 0,
                        MessageText := 'Command.Position.E2 = {1}',
                        Para1       :=  REAL_TO_STRING(_command.Position.E2));

// Create log entry for Position.E3
CreateLogMessagePara1 ( Timestamp   := AxesGroup.InternalData.SystemTime,
                        MessageType := MessageType.CMD,
                        Severity    := Severity.DEBUG,
                        MessageCode := 0,
                        MessageText := 'Command.Position.E3 = {1}',
                        Para1       :=  REAL_TO_STRING(_command.Position.E3));

// Create log entry for Position.E4
CreateLogMessagePara1 ( Timestamp   := AxesGroup.InternalData.SystemTime,
                        MessageType := MessageType.CMD,
                        Severity    := Severity.DEBUG,
                        MessageCode := 0,
                        MessageText := 'Command.Position.E4 = {1}',
                        Para1       :=  REAL_TO_STRING(_command.Position.E4));

// Create log entry for Position.E5
CreateLogMessagePara1 ( Timestamp   := AxesGroup.InternalData.SystemTime,
                        MessageType := MessageType.CMD,
                        Severity    := Severity.DEBUG,
                        MessageCode := 0,
                        MessageText := 'Command.Position.E5 = {1}',
                        Para1       :=  REAL_TO_STRING(_command.Position.E5));

// Create log entry for Position.E6
CreateLogMessagePara1 ( Timestamp   := AxesGroup.InternalData.SystemTime,
                        MessageType := MessageType.CMD,
                        Severity    := Severity.DEBUG,
                        MessageCode := 0,
                        MessageText := 'Command.Position.E6 = {1}',
                        Para1       :=  REAL_TO_STRING(_command.Position.E6));
END_METHOD

METHOD FB_init : BOOL
VAR_INPUT
  /// if TRUE, the retain variables are initialized (warm start / cold start)
  bInitRetains : BOOL; 
  /// if TRUE, the instance afterwards gets moved into the copy code (online change)
  bInCopyCode  : BOOL;  
END_VAR
MyType := 'MC_CalculateFrameFB';

ExecMode := ExecutionMode.PARALLEL;
END_METHOD

METHOD PROTECTED OnCall
VAR_IN_OUT
  /// Robot assignment of function
  AxesGroup : AxesGroup; 
END_VAR
// call base implementation
SUPER^.OnCall(AxesGroup := AxesGroup);

CASE _stepCmd OF
  
  00:  IF ( _execute_R.Q )  
       THEN
         // Check function is supported and parameter are valid ?
         IF (( CheckFunctionSupported( AxesGroup := AxesGroup )) AND
             ( CheckParameterValid   ( AxesGroup := AxesGroup )))      
         THEN
           // set busy flag
           Busy := TRUE;
           // Reset command outputs
           SysDepMemSet(pDest := ADR(OutCmd), Value := 0, DataLen := SIZEOF(OutCmd));         
           // apply command parameter
          _parCmd := ParCmd;
           // init parameter sequence
          _command.ParSeq := 1;
           // set timeout
           SetTimeout(PT := _timeoutCmd, rTimer := _timerCmd);
           // inc step counter
          _stepCmd := _stepCmd + 1; 
         END_IF
       END_IF
     

  01: // inc data index 
     _dataIndex := _dataIndex + 1;

      CASE _parCmd.Mode OF
        FrameCalculationMode.ONE_POINT_METHOD   :
          _dataComplete := _dataIndex >= 1;
        FrameCalculationMode.THREE_POINT_METHOD :
          _dataComplete := _dataIndex >= 3;
        FrameCalculationMode.FOUR_POINT_METHOD  :
          _dataComplete := _dataIndex >= 4; 
      END_CASE

       // create command data
       CommandData := CreateCommandPayload(AxesGroup := AxesGroup);
       // Add command to active command register
      _uniqueID := AxesGroup.Acyclic.ActiveCommandRegister.AddCmd( pCommandFB := ADR(THIS^ ));     
       // set timeout
       SetTimeout(PT := _timeoutCmd, rTimer := _timerCmd);
       // inc step counter
      _stepCmd := _stepCmd + 1; 


  02:  // Wait for responce received
       IF ( _responseReceived )
       THEN
         // reset response received flag
        _responseReceived := FALSE;

         CASE  _response.State 
         OF
           CmdMessageState.BUFFERED : CommandBuffered := TRUE;
           CmdMessageState.DONE     : Done            := TRUE;
           CmdMessageState.ERROR    : Error           := TRUE;
         END_CASE
                
         // Done, Aborted or Error ?
         IF (_response.State >= CmdMessageState.DONE )
         THEN
           // Reset Busy Flag
           Busy := FALSE;
           // Update results
           OutCmd.IEC_Date       := _response.IEC_Date;
           OutCmd.IEC_TIME       := _response.IEC_TIME;
           OutCmd.ReferenceFrame := _response.ReferenceFrame;
           OutCmd.Position       := _response.Position;

           IF ( _dataComplete ) OR (_response.State = CmdMessageState.ABORTED )
           THEN
             // set timeout
             SetTimeout(PT := _timeoutCmd, rTimer := _timerCmd);
             // inc step counter
            _stepCmd := _stepCmd + 1; 
           ELSE
             // set timeout
             SetTimeout(PT := _timeoutCmd, rTimer := _timerCmd);
             // dec step counter
            _stepCmd := _stepCmd - 1; 
           END_IF
         END_IF
       END_IF


  03: IF ( NOT Execute)
      THEN
        Reset();
      END_IF     
      
ELSE
  // invalid step
  ErrorID := RobotLibraryEvents.ERR_INVALID_STEP;
END_CASE


// Reset FB
IF ( NOT Execute )
THEN
  Reset();
END_IF
END_METHOD

METHOD INTERNAL ParseResponsePayload : DINT
VAR_INPUT
  /// Response data
  ResponseData : RobotLibraryRecvDataFB;
  /// Timestamp
  Timestamp    : SystemTime;  
END_VAR
// Table 6-657: Received CMD payload (RC to PLC) of "CalculateFrame"
// --------------------------
// Header
// --------------------------
// Byte 00 : USINT     - ParSeq | State     
// Byte 01 : SINT      - AlarmMessageSeverity    
// Byte 02 : UINT      - AlarmMessageCode HB
// Byte 03 :           - AlarmMessageCode LB
// --------------------------
// Datablock
// --------------------------
// Byte 04 : IEC_DATE  - FrameData.Date HB
// Byte 05 :           - FrameData.Date LB
// Byte 06 : IEC_TIME  - FrameData.Time HB HW
// Byte 07 :           - FrameData.Time HB LW
// Byte 08 :           - FrameData.Time LW HB
// Byte 09 :           - FrameData.Time LW LB
// Byte 10 : USINT     - FrameData.ReferenceFrame
// Byte 11 : BYTE      - Reserve
// Byte 12 : REAL      - FrameData.X  HB HW
// Byte 13 :           - FrameData.X  HB LW
// Byte 14 :           - FrameData.X  LW HB
// Byte 15 :           - FrameData.X  LW LB
// Byte 16 : REAL      - FrameData.Y  HB HW
// Byte 17 :           - FrameData.Y  HB LW
// Byte 18 :           - FrameData.Y  LW HB
// Byte 19 :           - FrameData.Y  LW LB
// Byte 20 : REAL      - FrameData.Z  HB HW
// Byte 21 :           - FrameData.Z  HB LW
// Byte 22 :           - FrameData.Z  LW HB
// Byte 23 :           - FrameData.Z  LW LB
// Byte 24 : REAL      - FrameData.Rx HB HW
// Byte 25 :           - FrameData.Rx HB LW
// Byte 26 :           - FrameData.Rx LW HB
// Byte 27 :           - FrameData.Rx LW LB
// Byte 28 : REAL      - FrameData.Ry HB HW
// Byte 29 :           - FrameData.Ry HB LW
// Byte 30 :           - FrameData.Ry LW HB
// Byte 31 :           - FrameData.Ry LW LB
// Byte 32 : REAL      - FrameData.Rz HB HW
// Byte 33 :           - FrameData.Rz HB LW
// Byte 34 :           - FrameData.Rz LW HB
// Byte 35 :           - FrameData.Rz LW LB
// --------------------------
// call base implementation to parse the header from payload buffer
ResponseData.PayloadPtr := SUPER^.ParseResponsePayload(ResponseData := ResponseData, Timestamp := Timestamp);

// copy parsed header to response
_response.ParSeq               := _rspHeader.ParSeq;
_response.State                := _rspHeader.State;
_response.AlarmMessageSeverity := _rspHeader.AlarmMessageSeverity;
_response.AlarmMessageCode     := _rspHeader.AlarmMessageCode;

// Get response.IEC_Date
_response.IEC_Date   := ResponseData.GetIecDate();
// Get response.IEC_TIME
_response.IEC_TIME   := ResponseData.GetIecTime();
// Get response.ReferenceFrame
_response.ReferenceFrame := ResponseData.GetUsint();
// Get response.Reserve
_response.Reserve := ResponseData.GetByte();
// Get response.Position.X
_response.Position.X := ResponseData.GetReal();
// Get response.Position.Y
_response.Position.Y := ResponseData.GetReal();
// Get response.Position.Z
_response.Position.Z := ResponseData.GetReal();
// Get response.Position.Rx
_response.Position.Rx := ResponseData.GetReal();
// Get response.Position.Ry
_response.Position.Ry := ResponseData.GetReal();
// Get response.Position.Rz
_response.Position.Rz := ResponseData.GetReal();

// Create logging
ParseResponsePayloadLog(ResponseData := ResponseData, Timestamp := Timestamp);
END_METHOD

METHOD INTERNAL ParseResponsePayloadLog
VAR_INPUT
  /// Response data
  ResponseData : RobotLibraryRecvDataFB;
  /// Timestamp
  Timestamp    : SystemTime;  
END_VAR
// Create log entry for Parameter start
CreateLogMessage      ( Timestamp   := Timestamp,
                        MessageType := MessageType.CMD,
                        Severity    := Severity.DEBUG,
                        MessageCode := 0,
                        MessageText := 'Parsed the following parameter(s) from response data:');

// Create log entry for IEC_Date
CreateLogMessagePara1 ( Timestamp   := Timestamp,
                        MessageType := MessageType.CMD,
                        Severity    := Severity.DEBUG,
                        MessageCode := 0,
                        MessageText := 'Response.IEC_Date = {1}',
                        Para1       :=  IEC_DATE_TO_STRING(_response.IEC_Date));

// Create log entry for IEC_TIME
CreateLogMessagePara1 ( Timestamp   := Timestamp,
                        MessageType := MessageType.CMD,
                        Severity    := Severity.DEBUG,
                        MessageCode := 0,
                        MessageText := 'Response.IEC_TIME = {1}',
                        Para1       :=  IEC_TIME_TO_STRING(_response.IEC_TIME));

// Create log entry for ReferenceFrame
CreateLogMessagePara1 ( Timestamp   := Timestamp,
                        MessageType := MessageType.CMD,
                        Severity    := Severity.DEBUG,
                        MessageCode := 0,
                        MessageText := 'Response.ReferenceFrame = {1}',
                        Para1       :=  USINT_TO_STRING(_response.ReferenceFrame));

// Create log entry for Reserve
CreateLogMessagePara1 ( Timestamp   := Timestamp,
                        MessageType := MessageType.CMD,
                        Severity    := Severity.DEBUG,
                        MessageCode := 0,
                        MessageText := 'Response.Reserve = {1}',
                        Para1       :=  BYTE_TO_STRING(_response.Reserve));

// Create log entry for Position.X
CreateLogMessagePara1 ( Timestamp   := Timestamp,
                        MessageType := MessageType.CMD,
                        Severity    := Severity.DEBUG,
                        MessageCode := 0,
                        MessageText := 'Response.Position.X = {1}',
                        Para1       :=  REAL_TO_STRING(_response.Position.X));

// Create log entry for Position.Y
CreateLogMessagePara1 ( Timestamp   := Timestamp,
                        MessageType := MessageType.CMD,
                        Severity    := Severity.DEBUG,
                        MessageCode := 0,
                        MessageText := 'Response.Position.Y = {1}',
                        Para1       :=  REAL_TO_STRING(_response.Position.Y));

// Create log entry for Position.Z
CreateLogMessagePara1 ( Timestamp   := Timestamp,
                        MessageType := MessageType.CMD,
                        Severity    := Severity.DEBUG,
                        MessageCode := 0,
                        MessageText := 'Response.Position.Z = {1}',
                        Para1       :=  REAL_TO_STRING(_response.Position.Z));

// Create log entry for Position.Rx
CreateLogMessagePara1 ( Timestamp   := Timestamp,
                        MessageType := MessageType.CMD,
                        Severity    := Severity.DEBUG,
                        MessageCode := 0,
                        MessageText := 'Response.Position.Rx = {1}',
                        Para1       :=  REAL_TO_STRING(_response.Position.Rx));

// Create log entry for Position.Ry
CreateLogMessagePara1 ( Timestamp   := Timestamp,
                        MessageType := MessageType.CMD,
                        Severity    := Severity.DEBUG,
                        MessageCode := 0,
                        MessageText := 'Response.Position.Ry = {1}',
                        Para1       :=  REAL_TO_STRING(_response.Position.Ry));

// Create log entry for Position.Rz
CreateLogMessagePara1 ( Timestamp   := Timestamp,
                        MessageType := MessageType.CMD,
                        Severity    := Severity.DEBUG,
                        MessageCode := 0,
                        MessageText := 'Response.Position.Rz = {1}',
                        Para1       :=  REAL_TO_STRING(_response.Position.Rz));
END_METHOD

METHOD PROTECTED Reset : DINT
VAR_INPUT
END_VAR
Reset := SUPER^.Reset();

Done               := FALSE;
Busy               := FALSE;
CommandBuffered    := FALSE;
END_METHOD

END_FUNCTION_BLOCK

// Library/POUs/Calculation/MC_CalculateInverseKinematic/MC_CalculateInverseKinematicFB
/// Calculate Inverse Kinematic
FUNCTION_BLOCK MC_CalculateInverseKinematicFB EXTENDS RobotLibraryBaseExecuteFB
// ------------------------------------------------------------------------- 
//  SRCI Robot Library                                                
// ------------------------------------------------------------------------- 
//                                                                           
//  Object:      CalculateInverseKinematicFB                                       
//  Author:      Thorsten Brach                                                
//  Date:        2024-06-09
//
//  Description:                                              
//   
//                                                                           
//  Copyright: 
//    (C) 2024 Thorsten Brach. All rights reserved                                                                                                                                            
//             Licensed under the LGPL-3.0 license.
//                                                                           
//  Disclaimer:                                                                           
//    This project is provided without any guarantee and can be used for   
//    private and commercial purposes. Any use is at the user’s 
//    own risk and responsibility.
//
// -------------------------------------------------------------------------
VAR_INPUT
  /// Command parameter 
  ParCmd          : CalculateInverseKinematicParCmd;    
END_VAR
VAR_OUTPUT
  CommandBuffered : BOOL;
  /// Command output 
  OutCmd          : CalculateInverseKinematicOutCmd;  
END_VAR

VAR
  /// internal copy of command parameter 
 _parCmd          : CalculateInverseKinematicParCmd;
  /// command data to send
 _command         : CalculateInverseKinematicSendData;
  /// response data received
 _response        : CalculateInverseKinematicRecvData;      
END_VAR

SUPER^(AxesGroup := AxesGroup);

METHOD PROTECTED CheckFunctionSupported : BOOL
VAR_IN_OUT
  /// Robot assignment of function
  AxesGroup : AxesGroup; 
END_VAR
CheckFunctionSupported := AxesGroup.InternalData.RCSupportedFunctions.CalculateInverseKinematic;

IF ( NOT CheckFunctionSupported )
THEN
  // call base implementation for set error and create log entry
  SUPER^.CheckFunctionSupported(AxesGroup := AxesGroup);
END_IF
END_METHOD

METHOD PROTECTED CheckParameterChanged : BOOL
VAR_IN_OUT
  /// Robot assignment of function
  AxesGroup    : AxesGroup; 
END_VAR
// Check ParCmd Size is > 0, because MemCmp does not work correctly with size = 0
IF (SIZEOF(ParCmd) = 0) 
THEN 
  RETURN;
END_IF

// compare memory 
_parameterChanged := ( SysDepMemCmp(pData1 := ADR(ParCmd), pData2 := ADR(_parCmd), DataLen := SIZEOF(ParCmd)) <> RobotLibraryConstants.OK );

// check parameter valid ?
_parameterValid   := CheckParameterValid( AxesGroup := AxesGroup );

IF ((  _parameterChanged        )  AND 
    (  _parameterValid          )) OR
    (  _parameterUpdateInternal )  
THEN  
  // reset internal flag for send parameter update
 _parameterUpdateInternal := FALSE;
  // update internal copy of parameters 
 _parCmd := ParCmd;
  // inc parameter sequence
 _command.ParSeq := _command.ParSeq + 1;
  // update command data  
  CommandData := CreateCommandPayload(AxesGroup := AxesGroup); // ( Access via reference to rCommandFB in ACR )
  // notify active command register 
  AxesGroup.Acyclic.ActiveCommandRegister.NotifyParameterChanged := _uniqueID;
END_IF
END_METHOD

METHOD INTERNAL CreateCommandPayload : RobotLibrarySendDataFB
VAR_IN_OUT
  /// Robot assignment of function
  AxesGroup : AxesGroup; 
END_VAR
// Table 6-638: Sent CMD payload (PLC to RC) of "CalculateInverseKinematic"
// --------------------------
// Header
// --------------------------
// Byte 00 : UINT       - Type HB     
// Byte 01 :            - Type LB    
// Byte 02 : USINT      - Reserve | ExecutionMode
// Byte 03 : USINT      - ParSeq  | Priority
// --------------------------
// Datablock
// --------------------------
// Byte 04 : USINT      - ToolNo
// Byte 05 : USINT      - FrameNo
// Byte 06 : REAL       - Position.X  HW HB
// Byte 07 :            - Position.X  HW LB
// Byte 08 :            - Position.X  LW HB
// Byte 09 :            - Position.X  LW LB
// Byte 10 : REAL       - Position.Y  HW HB
// Byte 11 :            - Position.Y  HW LB
// Byte 12 :            - Position.Y  LW HB
// Byte 13 :            - Position.Y  LW LB
// Byte 14 : REAL       - Position.Z  HW HB
// Byte 15 :            - Position.Z  HW LB
// Byte 16 :            - Position.Z  LW HB
// Byte 17 :            - Position.Z  LW LB
// Byte 18 : REAL       - Position.Rx HW HB
// Byte 19 :            - Position.Rx HW LB
// Byte 20 :            - Position.Rx LW HB
// Byte 21 :            - Position.Rx LW LB
// Byte 22 : REAL       - Position.Ry HW HB
// Byte 23 :            - Position.Ry HW LB
// Byte 24 :            - Position.Ry LW HB
// Byte 25 :            - Position.Ry LW LB
// Byte 26 : REAL       - Position.Rz HW HB
// Byte 27 :            - Position.Rz HW LB
// Byte 28 :            - Position.Rz LW HB
// Byte 29 :            - Position.Rz LW LB
// Byte 30 : Config     - ArmConfig   LW HB
// Byte 31 :            - ArmConfig   LW LB
// Byte 32 : TurnNumber - J1 + J2     LW HB
// Byte 33 :            - J3 + J4     LW LB
// Byte 34 :            - J5 + J6     LW LB
// Byte 35 :            - E1          LW LB
// Byte 36 : REAL       - Position.E1 HW HB
// Byte 37 :            - Position.E1 HW LB
// Byte 38 :            - Position.E1 LW HB
// Byte 39 :            - Position.E1 LW LB
// Byte 40 : REAL       - Position.E2 HW HB
// Byte 41 :            - Position.E2 HW LB
// Byte 42 :            - Position.E2 LW HB
// Byte 43 :            - Position.E2 LW LB
// Byte 44 : REAL       - Position.E3 HW HB
// Byte 45 :            - Position.E3 HW LB
// Byte 46 :            - Position.E3 LW HB
// Byte 47 :            - Position.E3 LW LB
// Byte 48 : REAL       - Position.E4 HW HB
// Byte 49 :            - Position.E4 HW LB
// Byte 50 :            - Position.E4 LW HB
// Byte 51 :            - Position.E4 LW LB
// Byte 52 : REAL       - Position.E5 HW HB
// Byte 53 :            - Position.E5 HW LB
// Byte 54 :            - Position.E5 LW HB
// Byte 55 :            - Position.E5 LW LB
// Byte 56 : REAL       - Position.E6 HW HB
// Byte 57 :            - Position.E6 HW LB
// Byte 58 :            - Position.E6 LW HB
// Byte 59 :            - Position.E6 LW LB
// --------------------------
// set command parameter 
_command.CmdTyp            :=  CmdType.CalculateInverseKinematic;
_command.ExecMode          :=  ExecMode;
_command.ParSeq            := _command.ParSeq;
_command.Priority          :=  Priority;
_command.ToolNo            := _parCmd.ToolNo;
_command.FrameNo           := _parCmd.FrameNo;
_command.CartesianPosition := _parCmd.CartesianPosition;

// copy command data to header
_cmdHeader := _command;
// call base implementation to copy header to payload buffer
CreateCommandPayload := SUPER^.CreateCommandPayload(AxesGroup := AxesGroup);

// add command.TargetFrameNo
CreateCommandPayload.AddUsint(_command.ToolNo);
// add command.FrameNo
CreateCommandPayload.AddUsint(_command.FrameNo);
// add command.CartesianPosition.X
CreateCommandPayload.AddReal(_command.CartesianPosition.X);
// add command.CartesianPosition.Y
CreateCommandPayload.AddReal(_command.CartesianPosition.Y);
// add command.CartesianPosition.Z
CreateCommandPayload.AddReal(_command.CartesianPosition.Z);
// add command.CartesianPosition.Rx
CreateCommandPayload.AddReal(_command.CartesianPosition.Rx);
// add command.CartesianPosition.Ry
CreateCommandPayload.AddReal(_command.CartesianPosition.Ry);
// add command.CartesianPosition.Rz
CreateCommandPayload.AddReal(_command.CartesianPosition.Rz);
// add command.CartesianPosition.Config
CreateCommandPayload.AddArmConfig(_command.CartesianPosition.Config);
// add command.CartesianPosition.TurnNumber
CreateCommandPayload.AddTurnNumber(_command.CartesianPosition.TurnNumber);
// add command.CartesianPosition.E1
CreateCommandPayload.AddReal(_command.CartesianPosition.E1);
// add command.CartesianPosition.E2
CreateCommandPayload.AddReal(_command.CartesianPosition.E2);
// add command.CartesianPosition.E3
CreateCommandPayload.AddReal(_command.CartesianPosition.E3);
// add command.CartesianPosition.E4
CreateCommandPayload.AddReal(_command.CartesianPosition.E4);
// add command.CartesianPosition.E5
CreateCommandPayload.AddReal(_command.CartesianPosition.E5);
// add command.CartesianPosition.E6
CreateCommandPayload.AddReal(_command.CartesianPosition.E6);

// Create logging
CreateCommandPayloadLog(AxesGroup := AxesGroup);
END_METHOD

METHOD INTERNAL CreateCommandPayloadLog 
VAR_IN_OUT
  /// Robot assignment of function
  AxesGroup : AxesGroup; 
END_VAR
// Create log entry for Parameter start
CreateLogMessage      ( Timestamp   := AxesGroup.InternalData.SystemTime,
                        MessageType := MessageType.CMD,
                        Severity    := Severity.DEBUG,
                        MessageCode := 0,
                        MessageText := 'Create command payload with the following parameter(s) :');

// Create log entry for ToolNo
CreateLogMessagePara1 ( Timestamp   := AxesGroup.InternalData.SystemTime,
                        MessageType := MessageType.CMD,
                        Severity    := Severity.DEBUG,
                        MessageCode := 0,
                        MessageText := 'Command.ToolNo = {1}',
                        Para1       :=  USINT_TO_STRING(_command.ToolNo));

// Create log entry for FrameNo
CreateLogMessagePara1 ( Timestamp   := AxesGroup.InternalData.SystemTime,
                        MessageType := MessageType.CMD,
                        Severity    := Severity.DEBUG,
                        MessageCode := 0,
                        MessageText := 'Command.FrameNo = {1}',
                        Para1       :=  USINT_TO_STRING(_command.FrameNo));

// Create log entry for CartesianPosition.X
CreateLogMessagePara1 ( Timestamp   := AxesGroup.InternalData.SystemTime,
                        MessageType := MessageType.CMD,
                        Severity    := Severity.DEBUG,
                        MessageCode := 0,
                        MessageText := 'Command.CartesianPosition.X = {1}',
                        Para1       :=  REAL_TO_STRING(_command.CartesianPosition.X));

// Create log entry for CartesianPosition.Y
CreateLogMessagePara1 ( Timestamp   := AxesGroup.InternalData.SystemTime,
                        MessageType := MessageType.CMD,
                        Severity    := Severity.DEBUG,
                        MessageCode := 0,
                        MessageText := 'Command.CartesianPosition.Y = {1}',
                        Para1       :=  REAL_TO_STRING(_command.CartesianPosition.Y));

// Create log entry for CartesianPosition.Z
CreateLogMessagePara1 ( Timestamp   := AxesGroup.InternalData.SystemTime,
                        MessageType := MessageType.CMD,
                        Severity    := Severity.DEBUG,
                        MessageCode := 0,
                        MessageText := 'Command.CartesianPosition.Z = {1}',
                        Para1       :=  REAL_TO_STRING(_command.CartesianPosition.Z));

// Create log entry for CartesianPosition.Rx
CreateLogMessagePara1 ( Timestamp   := AxesGroup.InternalData.SystemTime,
                        MessageType := MessageType.CMD,
                        Severity    := Severity.DEBUG,
                        MessageCode := 0,
                        MessageText := 'Command.CartesianPosition.Rx = {1}',
                        Para1       :=  REAL_TO_STRING(_command.CartesianPosition.Rx));

// Create log entry for CartesianPosition.Ry
CreateLogMessagePara1 ( Timestamp   := AxesGroup.InternalData.SystemTime,
                        MessageType := MessageType.CMD,
                        Severity    := Severity.DEBUG,
                        MessageCode := 0,
                        MessageText := 'Command.CartesianPosition.Ry = {1}',
                        Para1       :=  REAL_TO_STRING(_command.CartesianPosition.Ry));

// Create log entry for CartesianPosition.Rz
CreateLogMessagePara1 ( Timestamp   := AxesGroup.InternalData.SystemTime,
                        MessageType := MessageType.CMD,
                        Severity    := Severity.DEBUG,
                        MessageCode := 0,
                        MessageText := 'Command.CartesianPosition.Rz = {1}',
                        Para1       :=  REAL_TO_STRING(_command.CartesianPosition.Rz));

// Create log entry for CartesianPosition.Config
CreateLogMessagePara1 ( Timestamp   := AxesGroup.InternalData.SystemTime,
                        MessageType := MessageType.CMD,
                        Severity    := Severity.DEBUG,
                        MessageCode := 0,
                        MessageText := 'Command.CartesianPosition.Config = {1}',
                        Para1       :=  ARM_CONFIG_TO_STRING(_command.CartesianPosition.Config));

// Create log entry for CartesianPosition.TurnNumber[0]
CreateLogMessagePara1 ( Timestamp   := AxesGroup.InternalData.SystemTime,
                        MessageType := MessageType.CMD,
                        Severity    := Severity.DEBUG,
                        MessageCode := 0,
                        MessageText := 'Command.CartesianPosition.TurnNumber[0] = {1}',
                        Para1       :=  BYTE_TO_STRING(CombineHalfSints(HalfSintHi := _command.CartesianPosition.TurnNumber.J2Turns, 
                                                                        HalfSintLo := _command.CartesianPosition.TurnNumber.J1Turns)));

// Create log entry for CartesianPosition.TurnNumber[1]
CreateLogMessagePara1 ( Timestamp   := AxesGroup.InternalData.SystemTime,
                        MessageType := MessageType.CMD,
                        Severity    := Severity.DEBUG,
                        MessageCode := 0,
                        MessageText := 'Command.CartesianPosition.TurnNumber[1] = {1}',
                        Para1       :=  BYTE_TO_STRING(CombineHalfSints(HalfSintHi := _command.CartesianPosition.TurnNumber.J4Turns, 
                                                                        HalfSintLo := _command.CartesianPosition.TurnNumber.J3Turns)));

// Create log entry for CartesianPosition.TurnNumber[2]
CreateLogMessagePara1 ( Timestamp   := AxesGroup.InternalData.SystemTime,
                        MessageType := MessageType.CMD,
                        Severity    := Severity.DEBUG,
                        MessageCode := 0,
                        MessageText := 'Command.CartesianPosition.TurnNumber[2] = {1}',
                        Para1       :=  BYTE_TO_STRING(CombineHalfSints(HalfSintHi := _command.CartesianPosition.TurnNumber.J6Turns, 
                                                                        HalfSintLo := _command.CartesianPosition.TurnNumber.J5Turns)));

// Create log entry for CartesianPosition.TurnNumber[3]
CreateLogMessagePara1 ( Timestamp   := AxesGroup.InternalData.SystemTime,
                        MessageType := MessageType.CMD,
                        Severity    := Severity.DEBUG,
                        MessageCode := 0,
                        MessageText := 'Command.CartesianPosition.TurnNumber[3] = {1}',
                        Para1       :=  SINT_TO_STRING(_command.CartesianPosition.TurnNumber.E1Turns));

// Create log entry for CartesianPosition.E1
CreateLogMessagePara1 ( Timestamp   := AxesGroup.InternalData.SystemTime,
                        MessageType := MessageType.CMD,
                        Severity    := Severity.DEBUG,
                        MessageCode := 0,
                        MessageText := 'Command.CartesianPosition.E1 = {1}',
                        Para1       :=  REAL_TO_STRING(_command.CartesianPosition.E1));

// Create log entry for CartesianPosition.E2
CreateLogMessagePara1 ( Timestamp   := AxesGroup.InternalData.SystemTime,
                        MessageType := MessageType.CMD,
                        Severity    := Severity.DEBUG,
                        MessageCode := 0,
                        MessageText := 'Command.CartesianPosition.E2 = {1}',
                        Para1       :=  REAL_TO_STRING(_command.CartesianPosition.E2));

// Create log entry for CartesianPosition.E3
CreateLogMessagePara1 ( Timestamp   := AxesGroup.InternalData.SystemTime,
                        MessageType := MessageType.CMD,
                        Severity    := Severity.DEBUG,
                        MessageCode := 0,
                        MessageText := 'Command.CartesianPosition.E3 = {1}',
                        Para1       :=  REAL_TO_STRING(_command.CartesianPosition.E3));

// Create log entry for CartesianPosition.E4
CreateLogMessagePara1 ( Timestamp   := AxesGroup.InternalData.SystemTime,
                        MessageType := MessageType.CMD,
                        Severity    := Severity.DEBUG,
                        MessageCode := 0,
                        MessageText := 'Command.CartesianPosition.E4 = {1}',
                        Para1       :=  REAL_TO_STRING(_command.CartesianPosition.E4));

// Create log entry for CartesianPosition.E5
CreateLogMessagePara1 ( Timestamp   := AxesGroup.InternalData.SystemTime,
                        MessageType := MessageType.CMD,
                        Severity    := Severity.DEBUG,
                        MessageCode := 0,
                        MessageText := 'Command.CartesianPosition.E5 = {1}',
                        Para1       :=  REAL_TO_STRING(_command.CartesianPosition.E5));

// Create log entry for CartesianPosition.E6
CreateLogMessagePara1 ( Timestamp   := AxesGroup.InternalData.SystemTime,
                        MessageType := MessageType.CMD,
                        Severity    := Severity.DEBUG,
                        MessageCode := 0,
                        MessageText := 'Command.CartesianPosition.E6 = {1}',
                        Para1       :=  REAL_TO_STRING(_command.CartesianPosition.E6));
END_METHOD

